// TIA Portal V20 export
TYPE "LER_zp_CITICoS"
// stored: Access Published
   STRUCT
      Map_ID : SInt;   // Map ID
      Material_Low_Warning : Bool;   // Material Low Warning
      Auto_Cycle_Running : Bool;   // Auto Cycle Running
      Manual_Mode : Bool;   // Manual Mode
      Cycle_Time_Ready : Bool;   // Cycle Time Ready
      Overcycle : Bool;   // Overcycle
      OperatorOvercycle1 : Bool;   // Operator Overcycle 1
      OperatorOvercycle2 : Bool;   // Operator Overcycle 2
      Blocked : Bool;   // Blocked
      Starved : Bool;   // Starved
      Idle : Bool;   // Idle
      Wait_1 : Bool;   // Wait 1
      Wait_2 : Bool;   // Wait 2
      Wait_3 : Bool;   // Wait 3
      Wait_4 : Bool;   // Wait 4
      Stopped_by_Operator : Bool;   // Stopped by Operator
      Machine_Fault : Bool;   // Machine Fault
      Machine_Fault_Ack : Bool;   // Machine Fault Ack
      Quality_Check_Warning : Bool;   // Quality Check Warning
      Quality_Check_Fault : Bool;   // Quality Check Fault
      Quality_Check_Ack : Bool;   // Quality Check Ack
      Tool_Change_Warning : Bool;   // Tool Change Warning
      Tool_Change_Fault : Bool;   // Tool Change Fault
      Tool_Change_Ack : Bool;   // Tool Change Ack
      Spare_Bool_1 : Bool;
      Station_Andon_Hold : Bool;   // Station Andon Hold
      Filter_Minor_Fault : Bool;   // Filter Minor Fault
      Filter_Tank_Coolant_Temp_OK : Bool;   // Filter Tank Coolant Temp OK
      Filter_Tank_Coolant_Temp_High : Bool;   // Filter Tank Coolant Temp High
      Filter_Tank_Coolant_Temp_Low : Bool;   // Filter Tank Coolant Temp Low
      Filter_Tank_Level_OK : Bool;   // Filter Tank Level OK
      Filter_Tank_Level_High : Bool;   // Filter Tank Level High
      Filter_Tank_Level_Low : Bool;   // Filter Tank Level Low
      Filter_PumpBack_Level_OK : Bool;   // Filter Pump Back Level OK
      Filter_PumpBack_Level_High : Bool;   // Filter Pump Back Level High
      Filter_PumpBack_Level_Low : Bool;   // Filter Pump Back Level Low
      CMM_Bad_Quality_Data_Available : Bool;   // CMM Bad Quality Data Available
      CMM_No_Que_Available : Bool;   // CMM No Que Available
      CMM_Que_Available : Bool;   // CMM Que Available
      CMM_Inspection_Program_Running : Bool;   // CMM Inspection Program Running
      Spare_Bool_2 : Bool;
      CMM_Program_Minutes_Remaining : Int;   // CMM Program Minutes Remaining
      Date_of_Event : DInt;   // Date of Event
      Time_of_Event : DInt;   // Time of Event
      Fault_Word : DInt;   // Fault Word
   END_STRUCT;
END_TYPE
